Fanuc KAREL source: kf00076.KL

-- PROVISIONAL review KL for V770-1; original PC SHA256 0a195a1a3e897cb880ddd6d424d318c74a4881d545e72c85fffa8812ae6ab842
-- Incomplete behavior may be omitted. Consult companion uncertainty JSON. Do not deploy.
PROGRAM KF00076
%NOLOCKGROUP
BEGIN
  -- UNRESOLVED_PC offsets 5-15; opcodes 3F,75
  -- UNRESOLVED_PC offsets 20-29; opcodes 3F,75
  -- UNRESOLVED_PC offsets 34-45; opcodes 2E,23
  -- UNRESOLVED_PC offsets 50-61; opcodes 2E,23
  -- UNRESOLVED_PC offsets 66-96; opcodes 27,22,27,2E,27,2E,22,2A,31
  -- UNRESOLVED_PC offsets 101-105; opcodes 7F
END KF00076
